SUBAPPLICATION Uebung_019c (* Umschalten einer Maske *)
  (* Standard: 61499-2; Description: Copyright (c) 2023 Meisterschulen am Ostbahnhof This program and the accompanying materials are made available under the terms of the Eclipse Public License 2.0 which is available at https://www.eclipse.org/legal/epl-2.0/ SPDX-License-Identifier: EPL-2.0 *)
  (* Version 1.0, 2023-10-23, Franz Höpfinger, Meisterschulen am Ostbahnhof *)
  IMPORT logiBUS::io::DI::logiBUS_DI;
  IMPORT logiBUS::io::DQ::logiBUS_DO;
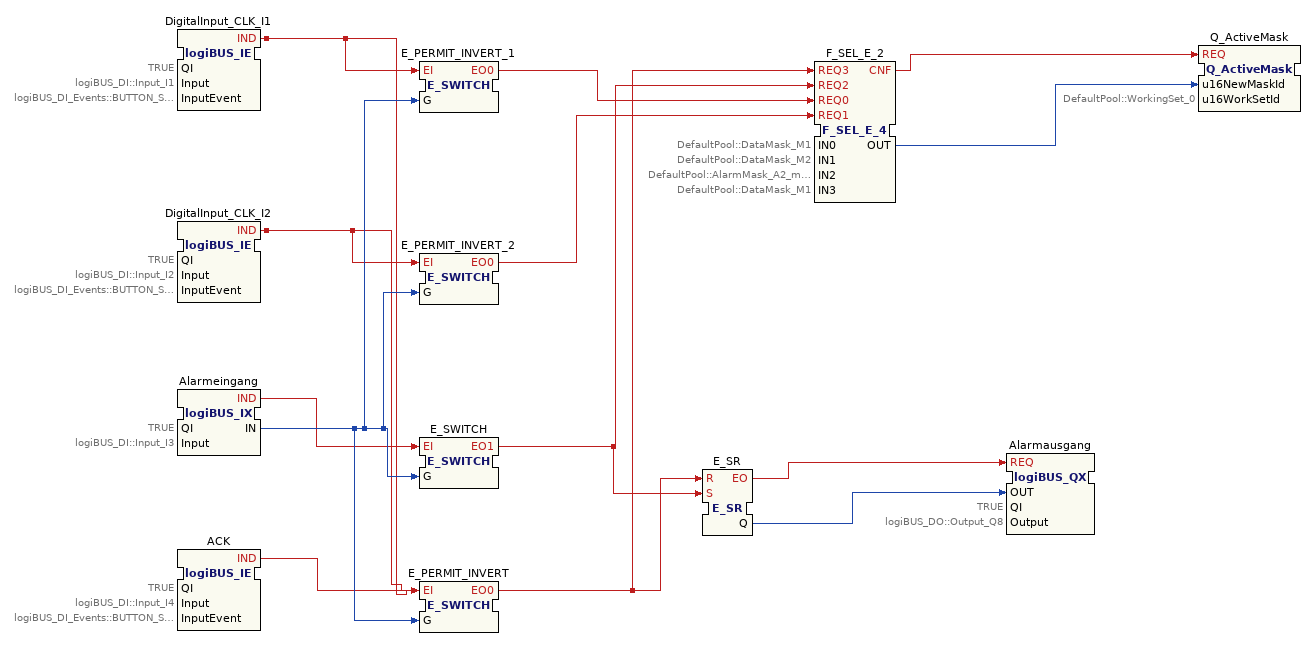
  FBS
    DigitalInput_CLK_I1 : logiBUS_IE(QI := TRUE, Input := logiBUS_DI::Input_I1, InputEvent := logiBUS_DI_Events::BUTTON_SINGLE_CLICK);
    Q_ActiveMask : isobus::ut::Q_ActiveMask(u16WorkSetId := DefaultPool::WorkingSet_0);
    DigitalInput_CLK_I2 : logiBUS_IE(QI := TRUE, Input := logiBUS_DI::Input_I2, InputEvent := logiBUS_DI_Events::BUTTON_SINGLE_CLICK);
    F_SEL_E_2 : F_SEL_E_4(IN0 := DefaultPool::DataMask_M1, IN1 := DefaultPool::DataMask_M2, IN2 := DefaultPool::AlarmMask_A2_medium, IN3 := DefaultPool::DataMask_M1);
    ACK : logiBUS_IE(QI := TRUE, Input := logiBUS_DI::Input_I4, InputEvent := logiBUS_DI_Events::BUTTON_SINGLE_CLICK);
    E_SR : iec61499::events::E_SR;
    Alarmausgang : logiBUS::io::DQ::logiBUS_QX(QI := TRUE, Output := logiBUS_DO::Output_Q8);
    Alarmeingang : logiBUS::io::DI::logiBUS_IX(QI := TRUE, Input := logiBUS_DI::Input_I3);
    E_SWITCH : iec61499::events::E_SWITCH;
    E_PERMIT_INVERT : iec61499::events::E_SWITCH;
    E_PERMIT_INVERT_1 : iec61499::events::E_SWITCH;
    E_PERMIT_INVERT_2 : iec61499::events::E_SWITCH;
  END_FBS
  EVENT_CONNECTIONS
    F_SEL_E_2.CNF TO Q_ActiveMask.REQ;
    E_PERMIT_INVERT.EO0 TO F_SEL_E_2.REQ3;
    E_PERMIT_INVERT.EO0 TO E_SR.R;
    E_SR.EO TO Alarmausgang.REQ;
    Alarmeingang.IND TO E_SWITCH.EI;
    E_SWITCH.EO1 TO F_SEL_E_2.REQ2;
    ACK.IND TO E_PERMIT_INVERT.EI;
    E_SWITCH.EO1 TO E_SR.S;
    DigitalInput_CLK_I1.IND TO E_PERMIT_INVERT.EI;
    DigitalInput_CLK_I2.IND TO E_PERMIT_INVERT.EI;
    DigitalInput_CLK_I1.IND TO E_PERMIT_INVERT_1.EI;
    DigitalInput_CLK_I2.IND TO E_PERMIT_INVERT_2.EI;
    E_PERMIT_INVERT_1.EO0 TO F_SEL_E_2.REQ0;
    E_PERMIT_INVERT_2.EO0 TO F_SEL_E_2.REQ1;
  END_CONNECTIONS
  DATA_CONNECTIONS
    F_SEL_E_2.OUT TO Q_ActiveMask.u16NewMaskId;
    E_SR.Q TO Alarmausgang.OUT;
    Alarmeingang.IN TO E_SWITCH.G;
    Alarmeingang.IN TO E_PERMIT_INVERT.G;
    Alarmeingang.IN TO E_PERMIT_INVERT_1.G;
    Alarmeingang.IN TO E_PERMIT_INVERT_2.G;
  END_CONNECTIONS
END_SUBAPPLICATION
